// TIA Portal project "Project1" (V21)

(* hardware
DEVICE "HMI_1"  TP700 Comfort
   slot 0: "HMI_1"  TP700 Comfort  6AV2 124-0GC01-0AX0  17.0.0.0
   slot 1: "HMI_RT_1"  TP700 Comfort  6AV2 124-0GC01-0AX0  17.0.0.0
   slot 5: "HMI_1.IE_CP_1"  PROFINET Interface  17.0.0.0
      slot 1: "PROFINET Interface_1"  PROFINET Interface
         slot 1: "Port_1"  Port
         slot 2: "Port_2"  Port
   slot 7: "HMI_1.MPI/DP_CP_1"  MPI/DP Interface  17.0.0.0
DEVICE "S7-1500/ET200MP station_1"  S7-1500 station
   slot 0: "Rail_0"  Rack  6ES7 590-1***0-0AA0
   slot 1: "PLC_1"  CPU 1515-2 PN  6ES7 515-2AM01-0AB0  V2.9
      slot 3: "CPU display_1"  6ES7591-1BA00-0AA0
      slot 32768: "PROFINET interface_1"  X1
         slot 32769: "Port_1"  X1 P1
         slot 32770: "Port_2"  X1 P2
      slot 33024: "PROFINET interface_2"  X2
         slot 33025: "Port_1"  X2 P1
      slot 34817: "Virtual CP interface port_1"  Virtual CP interface port  Virtual CP interface port
DEVICE "S7-1500/ET200MP station_2"  S7-1500 station
   slot 0: "Rail_0"  Rack  6ES7 590-1***0-0AA0
   slot 1: "PLC_2"  CPU 1515-2 PN  6ES7 515-2AN03-0AB0  V4.1
      slot 3: "CPU display_1"  6ES7591-1BA00-0AA0
      slot 32768: "PROFINET interface_1"  X1
         slot 32769: "Port_1"  X1 P1
         slot 32770: "Port_2"  X1 P2
      slot 33024: "PROFINET interface_2"  X2
         slot 33025: "Port_1"  X2 P1
      slot 34817: "Virtual CP interface port_1"  Virtual CP interface port  Virtual CP interface port FW V4.1
*)

// ===== PLC "PLC_1"  CPU 1515-2 PN =====

VAR_GLOBAL   // PLC tag table "Default tag table"
   "Bool_I0_0" AT %I0.0 : Bool;
   "Bool_I0_1" AT %I0.1 : Bool;
   "Bool_I1_5" AT %I1.5 : Bool;
   "Bool_Q0_0" AT %Q0.0 : Bool;
   "Bool_M0_1" AT %M0.1 : Bool;
   "Byte_IB2" AT %IB2 : Byte;
   "Byte_QB2" AT %QB2 : Byte;   // Датчик акустики, цех 1
   "Byte_MB11" AT %MB11 : Byte;
   "Char_IB3" AT %IB3 : Char;
   "Counter_C0" AT %C0 : Counter;
   "Date_IW4" AT %IW4 : Date;
   "Date_QW4" AT %QW4 : Date;
   "Date_MW12" AT %MW12 : Date;
   "DInt_ID6" AT %ID6 : DInt;
   "DInt_QD6" AT %QD50 : DInt;
   "DInt_MD14" AT %MD50 : DInt;
   "DWord_ID18" AT %ID18 : DWord;
   "DWord_QD22" AT %QD22 : DWord;
   "DWord_MD26" AT %MD26 : DWord;
   "Int_IW30" AT %IW30 : Int;
   "LDT_I32_0" AT %I32.0 : LDT;
   "LDT_Q40_0" AT %Q40.0 : LDT;
   "LDT_M48_0" AT %M48.0 : LDT;
   "LInt_M56_0" AT %M56.0 : LInt;
   "LReal_M64_0" AT %M64.0 : LReal;
   "LTime_I72_0" AT %I72.0 : LTime;
   "LTime_Q80_0" AT %Q80.0 : LTime;
   "LTime_M88_0" AT %M88.0 : LTime;
   "LTime_Of_Day_I96_0" AT %I96.0 : LTime_Of_Day;
   "LTime_Of_Day_Q104_0" AT %Q104.0 : LTime_Of_Day;
   "LTime_Of_Day_M112_0" AT %M112.0 : LTime_Of_Day;
   "LWord_M120_0" AT %M120.0 : LWord;
   "Real_MD128" AT %MD128 : Real;
   "S5Time_IW132" AT %IW132 : S5Time;
   "S5Time_QW134" AT %QW134 : S5Time;
   "S5Time_MW136" AT %MW136 : S5Time;
   "SInt_MB138" AT %MB138 : SInt;
   "Time_MD140" AT %MD140 : Time;
   "Time_Of_Day_MD144" AT %MD144 : Time_Of_Day;
   "Timer_T0" AT %T0 : Timer;
   "Timer_T1" AT %T1 : Timer;
   "UDInt_ID10" AT %ID10 : UDInt;
   "UInt_IW14" AT %IW14 : UInt;
   "ULInt_I22_0" AT %I22.0 : ULInt;
   "USInt_IB40" AT %IB40 : USInt;
   "WChar_IW42" AT %IW42 : WChar;
   "Word_IW44" AT %IW44 : Word;
   "Word_IW46" AT %IW46 : Word;
END_VAR

ORGANIZATION_BLOCK "Main"   // OB1, LAD, ProgramCycle
TITLE = "Main Program Sweep (Cycle)"
{ S7_Optimized_Access := 'TRUE' }
VERSION : 0.1
   VAR_INPUT
      Initial_Call : Bool;   // Initial call of this OB
      Remanence : Bool;   // =True, if remanent data are available
   END_VAR
BEGIN
END_ORGANIZATION_BLOCK

// ===== PLC "PLC_2"  CPU 1515-2 PN =====

VAR_GLOBAL   // PLC tag table "Default tag table"
   "vvvv" AT %I0.0 : Bool;
   "aaa" AT %IB1 : Char;
   "vvvv(1)" AT %ID5 : DInt;
END_VAR

ORGANIZATION_BLOCK "Main"   // OB1, LAD, ProgramCycle
TITLE = "Main Program Sweep (Cycle)"
{ S7_Optimized_Access := 'TRUE' }
VERSION : 0.1
   VAR_INPUT
      Initial_Call : Bool;   // Initial call of this OB
      Remanence : Bool;   // =True, if remanent data are available
   END_VAR
BEGIN
END_ORGANIZATION_BLOCK

(* ===== HMI "HMI_RT_1" =====
system functions are stored by id; their names below are inferred from use
connection "HMI_Connection_1": ETHERNET, S7_1500_OMS
connection "HMI_Connection_2": ETHERNET, S7_1500_OMS

HMI tags "Default tag table"
   "Tag_ScreenNumber" : UInt, internal
   "Tag_Int" : Int, internal
   "Bool" : Bool, internal
   "DateTime" : DateTime, internal
   "DInt" : DInt, internal
   "LReal" : LReal, internal
   "Real" : Real, internal
   "SInt" : SInt, internal
   "UDInt" : UDInt, internal
   "UInt" : UInt, internal
   "USInt" : USInt, internal
   "WString" : WString[254], internal
   "Array [0..22] of Bool" : Array [0..22] of Bool, internal
   "Array [0..22] of LReal" : Array [0..22] of LReal, internal
   "Array [5..22] of Int" : Array [0..22] of Int, internal
   "Array [0..22] of Bool_1" : Int, internal
   "AAAA" : WString[254], internal
   "xxxx" : Array [0..22] of UInt, internal
   "Bool_I0_0" : Bool = PLC Bool_I0_0 AT %I0.0, 1 s
   "Acoustic_Alarm" : Bool = PLC Bool_I0_1 AT %I0.1, 1 s
   "Bool_I1_5" : Bool = PLC Bool_I1_5 AT %I1.5, 1 s
   "Bool_Q0_0" : Bool = PLC Bool_Q0_0 AT %Q0.0, 1 s
   "Bool_M0_1" : Bool = PLC Bool_M0_1 AT %M0.1, 1 s
   "Byte_IB2" : Byte = PLC Byte_IB2 AT %IB2, 1 s
   "Byte_QB2" : Byte = PLC Byte_QB2 AT %QB2, 1 s
   "Byte_MB11" : Byte = PLC Byte_MB11 AT %MB11, 1 s
   "Char_IB3" : Char = PLC Char_IB3 AT %IB3, 1 s
   "Counter_C0" : Counter = PLC Counter_C0 AT %C0, 1 s
   "Date_IW4" : Date = PLC Date_IW4 AT %IW4, 1 s
   "Date_QW4" : Date = PLC Date_QW4 AT %QW4, 1 s   // Acoustic sensor level
   "Date_MW12" : Date = PLC Date_MW12 AT %MW12, 1 s   // Акустика: уровень шума, дБ
   "DInt_ID6" : DInt = PLC DInt_ID6 AT %ID6, 1 s
   "DInt_QD6" : DInt = PLC DInt_QD6 AT %QD50, 1 s
   "DInt_MD14" : DInt = PLC DInt_MD14 AT %MD50, 1 s
   "DWord_ID18" : DWord = PLC DWord_ID18 AT %ID18, 1 s
   "DWord_QD22" : DWord = PLC DWord_QD22 AT %QD22, 100 ms
   "DWord_MD26" : DWord = PLC DWord_MD26 AT %MD26, 10 s
   "Int_IW30" : Int = PLC Int_IW30 AT %IW30, 1 s
   "LDT_I32_0" : LDT = PLC LDT_I32_0 AT %I32.0, 1 s
   "LDT_Q40_0" : LDT = PLC LDT_Q40_0 AT %Q40.0, 1 s
   "LDT_M48_0" : LDT = PLC LDT_M48_0 AT %M48.0, 1 s
   "LInt_M56_0" : LInt = PLC LInt_M56_0 AT %M56.0, 1 s
   "LReal_M64_0" : LReal = PLC LReal_M64_0 AT %M64.0, 1 s
   "LTime_I72_0" : LTime = PLC LTime_I72_0 AT %I72.0, 1 s
   "LTime_Q80_0" : LTime = PLC LTime_Q80_0 AT %Q80.0, 1 s
   "LTime_M88_0" : LTime = PLC LTime_M88_0 AT %M88.0, 1 s
   "LTime_Of_Day_I96_0" : LTime_Of_Day = PLC LTime_Of_Day_I96_0 AT %I96.0, 1 s
   "LTime_Of_Day_Q104_0" : LTime_Of_Day = PLC LTime_Of_Day_Q104_0 AT %Q104.0, 1 s
   "LTime_Of_Day_M112_0" : LTime_Of_Day = PLC LTime_Of_Day_M112_0 AT %M112.0, 1 s
   "Real_MD128" : Real = PLC Real_MD128 AT %MD128, 1 s
   "S5Time_QW134" : S5Time = PLC S5Time_QW134 AT %QW134, 1 s   // Акустика: уровень шума, дБ
   "SInt_MB138" : SInt = PLC SInt_MB138 AT %MB138, 1 s
   "Time_MD140" : Time = PLC Time_MD140 AT %MD140, 1 s
   "Time_Of_Day_MD144" : Time_Of_Day = PLC Time_Of_Day_MD144 AT %MD144, 1 s
   "Timer_T0" : Timer = PLC Timer_T0 AT %T0, 1 s
   "Timer_T1" : Timer = PLC Timer_T1 AT %T1, 1 s
   "UDInt_ID10" : UDInt = PLC UDInt_ID10 AT %ID10, 1 s
   "UInt_IW14" : UInt = PLC UInt_IW14 AT %IW14, 1 s
   "ULInt_I22_0" : ULInt = PLC ULInt_I22_0 AT %I22.0, 1 s
   "USInt_IB40" : USInt = PLC USInt_IB40 AT %IB40, 1 s
   "WChar_IW42" : WChar = PLC WChar_IW42 AT %IW42, 1 s
   "Word_IW44" : Word = PLC Word_IW44 AT %IW44, 1 s
   "Word_IW46" : Word = PLC Word_IW46 AT %IW46, 1 s
   "xxxx_1" : Bool = PLC vvvv AT %I0.0, 1 s
   "xxxx_2" : Char = PLC aaa AT %IB1, 1 s
   "xxxx_3" : DInt = PLC "vvvv(1)" AT %ID5, 1 s

HMI tags "Tag table_1"
   "S5Time_MW136" : S5Time = PLC S5Time_MW136 AT %MW136, 1 s
   "S5Time_IW132" : S5Time = PLC S5Time_IW132 AT %IW132, 1 s

screen "Root screen" 800x420, template "Template_1"
   on GenerateScreen: SetTag("Tag_ScreenNumber", 1)
   TextField "HmiScreenItemData" at 80,166 size 640x25; Text 'Welcome to HMI_1 (TP700 Comfort)!'

Template "Template_1" 800x420
   Button "Exit" at 720,360 size 78x58; TextOff 'Exit'; PictureOff "ExitRuntime_TP700_Comfort_TR"; PictureOn "ExitRuntime_TP700_Comfort_TR"
      on Release: StopRuntime(0)
   Button "Template_Button" at 640,360 size 78x58; TextOff 'Text'
   Button "Template_Button_1" at 560,360 size 78x58; TextOff 'Text'
   Button "Template_Button_2" at 480,360 size 78x58; TextOff 'Text'
   Button "Template_Button_3" at 400,360 size 78x58; TextOff 'Text'
   Button "Template_Button_4" at 321,360 size 78x58; TextOff 'Text'
   Button "Template_Button_5" at 241,360 size 78x58; TextOff 'Text'
   Button "Template_Button_6" at 161,360 size 78x58; TextOff 'Text'
   Button "Alarms" at 81,360 size 78x58; TextOff 'Alarms'; PictureOff "AlarmDisplay_TP700_Comfort_TR"; PictureOn "AlarmDisplay_TP700_Comfort_TR"
      on Release: function_ef3f5d25("Alarm window_Unacknowledged", -1)
   Button "Start screen" at 1,360 size 78x58; TextOff 'Start screen'; PictureOff "NavigateHome_TP700_Comfort_TR"; PictureOn "NavigateHome_TP700_Comfort_TR"
      on Release: ActivateScreen("Root screen", 0)
*)